TYPE U_FLY_OPTIONS :
UNION

  stCtrl              : ARRAY[1..MAX_AXIS] OF ST_FLY_OPTIONS;

  byCtrl    AT %I*    : ARRAY[1..MAX_AXIS] OF
                        ARRAY[1..SIZEOF(ST_FLY_OPTIONS)] OF BYTE;

END_UNION
END_TYPE

(* stored: Version 1.1.0.1, ProductVersion 3.1.4026.18
   DUT U_FLY_OPTIONS: Id {a85a2647-4dc6-49fc-ad56-8f1f9ba259ba} *)
